// TIA Portal V20 export
DATA_BLOCK "RecipeParameter"   // DB168
// stored: MemoryReserve 100
   VAR
      unitRecipe : "LER_typeRecipe";
      ParameterSV { S7_SetPoint := 'True'} : "HMI_IF_Parameter_ListRecipe_UDT";
      ParameterPV { S7_SetPoint := 'True'} : "HMI_IF_Parameter_ListRecipe_UDT";
   END_VAR
BEGIN
   ParameterSV.Recipe6 := 9000000.0;
   ParameterSV.Recipe7 := 9000000.0;
   ParameterPV.Recipe6 := 300000.0;
   ParameterPV.Recipe7 := 300000.0;
END_DATA_BLOCK
